TYPE T_Sequence :
STRUCT
	pChild: POINTER TO fb_CtrlBase;
	// Access to CIF of child
	pCIF: POINTER TO T_Ctrl_CIf;
	// Associated run sequence group
	uinGroupRun: UINT;
	// Associated stop sequence group
	uinGroupStop: UINT;
	// Command to be executed for run sequence
	intCmdSeqRun: INT;
	// Expected status for run sequence
	intStatusSeqRun: INT;
	// Command to be executed for run sequence
	intCmdSeqStop: INT;
	// Expected status for run sequence
	intStatusSeqStop: INT;
END_STRUCT
END_TYPE

(* stored: Version 1.1.0.1, ProductVersion 3.1.0.19
   DUT T_Sequence: Id {9e110bfc-713a-494f-9c2a-36e36ac320de} *)
